TYPE FsT_MemArea : Tc2_System.E_TcMemoryArea; END_TYPE

(* stored: Version 1.1.0.1, ProductVersion 3.1.4024.4
   DUT FsT_MemArea: Id {8426e294-5de0-4837-a3bb-2a77f82ed5de} *)
